MoveL Offs(p0,121.96290000000002,30.827499999999997, 0), v100, z5, tool0;
MoveL Offs(p0,122.3,29.7, 0), v100, z5, tool0;
MoveL Offs(p0,121.74480000000001,29.45120000000001, 0), v100, z5, tool0;
MoveL Offs(p0,121.0427,29.323799999999995, 0), v100, z5, tool0;
MoveL Offs(p0,120.0904,29.197600000000005, 0), v100, z5, tool0;
MoveL Offs(p0,118.9125,29.075, 0), v100, z5, tool0;
MoveL Offs(p0,117.5336,28.9584, 0), v100, z5, tool0;
MoveL Offs(p0,115.97829999999999,28.8502, 0), v100, z5, tool0;
MoveL Offs(p0,114.2712,28.7528, 0), v100, z5, tool0;
MoveL Offs(p0,112.4369,28.668600000000005, 0), v100, z5, tool0;
MoveL Offs(p0,110.5,28.6, 0), v100, z5, tool0;
MoveL Offs(p0,103.26039999999998,28.309299999999997, 0), v100, z5, tool0;
MoveL Offs(p0,101.38480000000001,28.1456, 0), v100, z5, tool0;
MoveL Offs(p0,99.7,27.9375, 0), v100, z5, tool0;
MoveL Offs(p0,98.1592,27.6784, 0), v100, z5, tool0;
MoveL Offs(p0,96.7156,27.361699999999995, 0), v100, z5, tool0;
MoveL Offs(p0,95.32240000000002,26.9808, 0), v100, z5, tool0;
MoveL Offs(p0,93.9328,26.5291, 0), v100, z5, tool0;
MoveL Offs(p0,92.5,26.0, 0), v100, z5, tool0;
MoveL Offs(p0,91.52130000000001,25.629400000000004, 0), v100, z5, tool0;
MoveL Offs(p0,90.57440000000004,25.24320000000001, 0), v100, z5, tool0;
MoveL Offs(p0,89.6731,24.8498, 0), v100, z5, tool0;
MoveL Offs(p0,88.83120000000001,24.4576, 0), v100, z5, tool0;
MoveL Offs(p0,88.0625,24.075, 0), v100, z5, tool0;
MoveL Offs(p0,87.3808,23.7104, 0), v100, z5, tool0;
MoveL Offs(p0,86.79990000000001,23.3722, 0), v100, z5, tool0;
MoveL Offs(p0,86.3336,23.068800000000003, 0), v100, z5, tool0;
MoveL Offs(p0,85.99570000000001,22.808600000000002, 0), v100, z5, tool0;
MoveL Offs(p0,85.8,22.6, 0), v100, z5, tool0;
MoveL Offs(p0,85.14040000000001,22.216700000000003, 0), v100, z5, tool0;
MoveL Offs(p0,83.57879999999997,23.8249, 0), v100, z5, tool0;
MoveL Offs(p0,82.7536,25.5728, 0), v100, z5, tool0;
MoveL Offs(p0,81.95,27.7875, 0), v100, z5, tool0;
MoveL Offs(p0,81.2064,30.347199999999997, 0), v100, z5, tool0;
MoveL Offs(p0,80.56120000000001,33.130100000000006, 0), v100, z5, tool0;
MoveL Offs(p0,80.0528,36.0144, 0), v100, z5, tool0;
MoveL Offs(p0,79.7196,38.8783, 0), v100, z5, tool0;
MoveL Offs(p0,79.6,41.6, 0), v100, z5, tool0;
MoveL Offs(p0,80.06560000000002,47.246400000000015, 0), v100, z5, tool0;
MoveL Offs(p0,80.61339999999998,49.9151, 0), v100, z5, tool0;
MoveL Offs(p0,81.3808,52.49920000000001, 0), v100, z5, tool0;
MoveL Offs(p0,82.375,55.0125, 0), v100, z5, tool0;
MoveL Offs(p0,83.6032,57.46880000000001, 0), v100, z5, tool0;
MoveL Offs(p0,85.0726,59.88190000000001, 0), v100, z5, tool0;
MoveL Offs(p0,86.7904,62.265600000000006, 0), v100, z5, tool0;
MoveL Offs(p0,88.7638,64.6337, 0), v100, z5, tool0;
MoveL Offs(p0,91.0,67.0, 0), v100, z5, tool0;
MoveL Offs(p0,93.10790000000001,69.02610000000001, 0), v100, z5, tool0;
MoveL Offs(p0,95.17920000000002,70.84880000000001, 0), v100, z5, tool0;
MoveL Offs(p0,97.2253,72.4747, 0), v100, z5, tool0;
MoveL Offs(p0,99.2576,73.91040000000001, 0), v100, z5, tool0;
MoveL Offs(p0,101.2875,75.1625, 0), v100, z5, tool0;
MoveL Offs(p0,103.32639999999999,76.2376, 0), v100, z5, tool0;
MoveL Offs(p0,105.3857,77.1423, 0), v100, z5, tool0;
MoveL Offs(p0,107.4768,77.88320000000002, 0), v100, z5, tool0;
MoveL Offs(p0,109.6111,78.4669, 0), v100, z5, tool0;
MoveL Offs(p0,111.8,78.9, 0), v100, z5, tool0;
MoveL Offs(p0,114.63920000000005,79.21440000000003, 0), v100, z5, tool0;
MoveL Offs(p0,116.24330000000002,79.2951, 0), v100, z5, tool0;
MoveL Offs(p0,117.8816,79.3272, 0), v100, z5, tool0;
MoveL Offs(p0,119.4875,79.3125, 0), v100, z5, tool0;
MoveL Offs(p0,120.9944,79.25280000000001, 0), v100, z5, tool0;
MoveL Offs(p0,122.3357,79.1499, 0), v100, z5, tool0;
MoveL Offs(p0,124.7,78.6, 0), v100, z5, tool0;
MoveL Offs(p0,124.7,78.6, 0), v100, z5, tool0;
MoveJ Offs(p0,158.3,63.6, 10), v100, z1, tool0;
MoveL Offs(p0,158.5876,62.95320000000002, 0), v100, z5, tool0;
MoveL Offs(p0,158.84880000000007,62.33760000000001, 0), v100, z5, tool0;
MoveL Offs(p0,159.0812,61.76039999999999, 0), v100, z5, tool0;
MoveL Offs(p0,159.2824,61.2288, 0), v100, z5, tool0;
MoveL Offs(p0,159.45,60.75, 0), v100, z5, tool0;
MoveL Offs(p0,159.5816,60.3312, 0), v100, z5, tool0;
MoveL Offs(p0,159.6748,59.979600000000005, 0), v100, z5, tool0;
MoveL Offs(p0,159.7272,59.70240000000001, 0), v100, z5, tool0;
MoveL Offs(p0,159.7364,59.5068, 0), v100, z5, tool0;
MoveL Offs(p0,159.7,59.4, 0), v100, z5, tool0;
MoveL Offs(p0,158.64339999999999,59.0742, 0), v100, z5, tool0;
MoveL Offs(p0,157.9128,58.9104, 0), v100, z5, tool0;
MoveL Offs(p0,157.025,58.725, 0), v100, z5, tool0;
MoveL Offs(p0,155.9992,58.5216, 0), v100, z5, tool0;
MoveL Offs(p0,154.85459999999998,58.3038, 0), v100, z5, tool0;
MoveL Offs(p0,153.6104,58.07520000000001, 0), v100, z5, tool0;
MoveL Offs(p0,152.28580000000002,57.8394, 0), v100, z5, tool0;
MoveL Offs(p0,150.9,57.6, 0), v100, z5, tool0;
MoveL Offs(p0,147.34920000000002,57.077, 0), v100, z5, tool0;
MoveL Offs(p0,143.98560000000003,56.764000000000024, 0), v100, z5, tool0;
MoveL Offs(p0,140.8524,56.654999999999994, 0), v100, z5, tool0;
MoveL Offs(p0,137.99280000000002,56.74400000000001, 0), v100, z5, tool0;
MoveL Offs(p0,135.45,57.025, 0), v100, z5, tool0;
MoveL Offs(p0,131.4876,58.138999999999996, 0), v100, z5, tool0;
MoveL Offs(p0,130.1544,58.96, 0), v100, z5, tool0;
MoveL Offs(p0,129.3108,59.949, 0), v100, z5, tool0;
MoveL Offs(p0,129.0,61.1, 0), v100, z5, tool0;
MoveL Offs(p0,129.3213,61.807399999999994, 0), v100, z5, tool0;
MoveL Offs(p0,129.55360000000002,62.20880000000001, 0), v100, z5, tool0;
MoveL Offs(p0,129.8375,62.675, 0), v100, z5, tool0;
MoveL Offs(p0,130.1664,63.1952, 0), v100, z5, tool0;
MoveL Offs(p0,130.5337,63.7586, 0), v100, z5, tool0;
MoveL Offs(p0,130.9328,64.35440000000001, 0), v100, z5, tool0;
MoveL Offs(p0,131.3571,64.9718, 0), v100, z5, tool0;
MoveL Offs(p0,131.8,65.6, 0), v100, z5, tool0;
MoveL Offs(p0,132.95589999999999,67.0506, 0), v100, z5, tool0;
MoveL Offs(p0,134.25520000000006,68.45680000000002, 0), v100, z5, tool0;
MoveL Offs(p0,135.68529999999998,69.81020000000001, 0), v100, z5, tool0;
MoveL Offs(p0,137.23360000000002,71.10240000000002, 0), v100, z5, tool0;
MoveL Offs(p0,138.8875,72.325, 0), v100, z5, tool0;
MoveL Offs(p0,140.6344,73.4696, 0), v100, z5, tool0;
MoveL Offs(p0,142.4617,74.5278, 0), v100, z5, tool0;
MoveL Offs(p0,144.35680000000002,75.4912, 0), v100, z5, tool0;
MoveL Offs(p0,146.30710000000002,76.35140000000001, 0), v100, z5, tool0;
MoveL Offs(p0,148.3,77.1, 0), v100, z5, tool0;
MoveL Offs(p0,153.5,78.9, 0), v100, z5, tool0;
MoveL Offs(p0,155.1,73.2, 0), v100, z5, tool0;
MoveL Offs(p0,155.35970000000003,72.2346, 0), v100, z5, tool0;
MoveL Offs(p0,155.65360000000004,71.21280000000002, 0), v100, z5, tool0;
MoveL Offs(p0,155.9739,70.1562, 0), v100, z5, tool0;
MoveL Offs(p0,156.3128,69.0864, 0), v100, z5, tool0;
MoveL Offs(p0,156.6625,68.025, 0), v100, z5, tool0;
MoveL Offs(p0,157.0152,66.9936, 0), v100, z5, tool0;
MoveL Offs(p0,157.36309999999997,66.0138, 0), v100, z5, tool0;
MoveL Offs(p0,157.69840000000002,65.1072, 0), v100, z5, tool0;
MoveL Offs(p0,158.01330000000002,64.2954, 0), v100, z5, tool0;
MoveL Offs(p0,158.3,63.6, 0), v100, z5, tool0;
MoveL Offs(p0,158.3,63.6, 0), v100, z5, tool0;
MoveJ Offs(p0,118.3,63.5, 10), v100, z1, tool0;
MoveL Offs(p0,118.0768,57.86959999999999, 0), v100, z5, tool0;
MoveL Offs(p0,118.04589999999999,56.6078, 0), v100, z5, tool0;
MoveL Offs(p0,118.0216,55.31120000000001, 0), v100, z5, tool0;
MoveL Offs(p0,118.0057,54.001400000000004, 0), v100, z5, tool0;
MoveL Offs(p0,118.0,52.7, 0), v100, z5, tool0;
MoveL Offs(p0,117.9,44.9, 0), v100, z5, tool0;
MoveL Offs(p0,115.2,45.4, 0), v100, z5, tool0;
MoveL Offs(p0,113.98960000000004,45.60160000000002, 0), v100, z5, tool0;
MoveL Offs(p0,113.1804,45.7159, 0), v100, z5, tool0;
MoveL Offs(p0,112.26080000000002,45.83680000000001, 0), v100, z5, tool0;
MoveL Offs(p0,111.25,45.9625, 0), v100, z5, tool0;
MoveL Offs(p0,110.16720000000001,46.0912, 0), v100, z5, tool0;
MoveL Offs(p0,109.0316,46.2211, 0), v100, z5, tool0;
MoveL Offs(p0,107.86240000000001,46.3504, 0), v100, z5, tool0;
MoveL Offs(p0,106.6788,46.4773, 0), v100, z5, tool0;
MoveL Offs(p0,105.5,46.6, 0), v100, z5, tool0;
MoveL Offs(p0,100.6179,47.25800000000001, 0), v100, z5, tool0;
MoveL Offs(p0,96.65920000000001,48.192000000000014, 0), v100, z5, tool0;
MoveL Offs(p0,93.6353,49.372, 0), v100, z5, tool0;
MoveL Offs(p0,91.55760000000001,50.768, 0), v100, z5, tool0;
MoveL Offs(p0,90.4375,52.35, 0), v100, z5, tool0;
MoveL Offs(p0,90.28639999999999,54.088, 0), v100, z5, tool0;
MoveL Offs(p0,91.11569999999999,55.952, 0), v100, z5, tool0;
MoveL Offs(p0,92.9368,57.912, 0), v100, z5, tool0;
MoveL Offs(p0,95.7611,59.93800000000001, 0), v100, z5, tool0;
MoveL Offs(p0,99.6,62.0, 0), v100, z5, tool0;
MoveL Offs(p0,101.475,62.868600000000015, 0), v100, z5, tool0;
MoveL Offs(p0,103.41600000000001,63.66880000000002, 0), v100, z5, tool0;
MoveL Offs(p0,105.38699999999999,64.39219999999999, 0), v100, z5, tool0;
MoveL Offs(p0,107.35200000000002,65.03040000000001, 0), v100, z5, tool0;
MoveL Offs(p0,109.275,65.575, 0), v100, z5, tool0;
MoveL Offs(p0,111.12,66.0176, 0), v100, z5, tool0;
MoveL Offs(p0,112.851,66.3498, 0), v100, z5, tool0;
MoveL Offs(p0,114.43200000000002,66.56320000000001, 0), v100, z5, tool0;
MoveL Offs(p0,115.827,66.6494, 0), v100, z5, tool0;
MoveL Offs(p0,117.0,66.6, 0), v100, z5, tool0;
MoveL Offs(p0,117.74069999999999,66.2643, 0), v100, z5, tool0;
MoveL Offs(p0,117.91839999999999,66.04159999999999, 0), v100, z5, tool0;
MoveL Offs(p0,118.0625,65.7625, 0), v100, z5, tool0;
MoveL Offs(p0,118.1736,65.4264, 0), v100, z5, tool0;
MoveL Offs(p0,118.25230000000002,65.0327, 0), v100, z5, tool0;
MoveL Offs(p0,118.29920000000001,64.5808, 0), v100, z5, tool0;
MoveL Offs(p0,118.31490000000001,64.0701, 0), v100, z5, tool0;
MoveL Offs(p0,118.3,63.5, 0), v100, z5, tool0;
MoveL Offs(p0,118.3,63.5, 0), v100, z5, tool0;
MoveJ Offs(p0,77.2,61.7, 10), v100, z1, tool0;
MoveL Offs(p0,80.9,60.2, 0), v100, z5, tool0;
MoveL Offs(p0,78.9,55.1, 0), v100, z5, tool0;
MoveL Offs(p0,78.6038,54.2505, 0), v100, z5, tool0;
MoveL Offs(p0,78.31840000000001,53.39200000000002, 0), v100, z5, tool0;
MoveL Offs(p0,78.0486,52.5395, 0), v100, z5, tool0;
MoveL Offs(p0,77.7992,51.708000000000006, 0), v100, z5, tool0;
MoveL Offs(p0,77.575,50.9125, 0), v100, z5, tool0;
MoveL Offs(p0,77.3808,50.168, 0), v100, z5, tool0;
MoveL Offs(p0,77.22139999999999,49.4895, 0), v100, z5, tool0;
MoveL Offs(p0,77.1016,48.892, 0), v100, z5, tool0;
MoveL Offs(p0,77.02619999999999,48.39050000000001, 0), v100, z5, tool0;
MoveL Offs(p0,77.0,48.0, 0), v100, z5, tool0;
MoveL Offs(p0,76.732,46.63440000000001, 0), v100, z5, tool0;
MoveL Offs(p0,76.37899999999999,46.28009999999999, 0), v100, z5, tool0;
MoveL Offs(p0,75.864,46.147200000000005, 0), v100, z5, tool0;
MoveL Offs(p0,75.175,46.2375, 0), v100, z5, tool0;
MoveL Offs(p0,74.3,46.5528, 0), v100, z5, tool0;
MoveL Offs(p0,73.227,47.09490000000001, 0), v100, z5, tool0;
MoveL Offs(p0,70.439,48.8667, 0), v100, z5, tool0;
MoveL Offs(p0,68.7,50.1, 0), v100, z5, tool0;
MoveL Offs(p0,67.0042,51.4408, 0), v100, z5, tool0;
MoveL Offs(p0,65.46560000000002,52.810400000000016, 0), v100, z5, tool0;
MoveL Offs(p0,64.0974,54.1896, 0), v100, z5, tool0;
MoveL Offs(p0,62.91279999999999,55.5592, 0), v100, z5, tool0;
MoveL Offs(p0,61.925,56.9, 0), v100, z5, tool0;
MoveL Offs(p0,61.1472,58.1928, 0), v100, z5, tool0;
MoveL Offs(p0,60.59259999999999,59.4184, 0), v100, z5, tool0;
MoveL Offs(p0,60.2744,60.5576, 0), v100, z5, tool0;
MoveL Offs(p0,60.205799999999996,61.5912, 0), v100, z5, tool0;
MoveL Offs(p0,60.4,62.5, 0), v100, z5, tool0;
MoveL Offs(p0,60.80080000000002,63.24960000000002, 0), v100, z5, tool0;
MoveL Offs(p0,61.10920000000001,63.5179, 0), v100, z5, tool0;
MoveL Offs(p0,61.51840000000001,63.7208, 0), v100, z5, tool0;
MoveL Offs(p0,62.05,63.8625, 0), v100, z5, tool0;
MoveL Offs(p0,62.7256,63.947199999999995, 0), v100, z5, tool0;
MoveL Offs(p0,63.5668,63.9791, 0), v100, z5, tool0;
MoveL Offs(p0,64.5952,63.9624, 0), v100, z5, tool0;
MoveL Offs(p0,65.8324,63.901300000000006, 0), v100, z5, tool0;
MoveL Offs(p0,67.3,63.8, 0), v100, z5, tool0;
MoveL Offs(p0,69.44320000000002,63.55280000000001, 0), v100, z5, tool0;
MoveL Offs(p0,70.55980000000001,63.3842, 0), v100, z5, tool0;
MoveL Offs(p0,71.67760000000001,63.19040000000001, 0), v100, z5, tool0;
MoveL Offs(p0,72.775,62.975, 0), v100, z5, tool0;
MoveL Offs(p0,73.8304,62.74159999999999, 0), v100, z5, tool0;
MoveL Offs(p0,74.8222,62.4938, 0), v100, z5, tool0;
MoveL Offs(p0,75.7288,62.235200000000006, 0), v100, z5, tool0;
MoveL Offs(p0,76.52860000000001,61.96939999999999, 0), v100, z5, tool0;
MoveL Offs(p0,77.2,61.7, 0), v100, z5, tool0;
MoveL Offs(p0,77.2,61.7, 0), v100, z5, tool0;
MoveJ Offs(p0,252.7,48.8, 10), v100, z1, tool0;
MoveL Offs(p0,252.4381,48.368900000000004, 0), v100, z5, tool0;
MoveL Offs(p0,252.35920000000002,48.348800000000004, 0), v100, z5, tool0;
MoveL Offs(p0,252.2875,48.3875, 0), v100, z5, tool0;
MoveL Offs(p0,252.22479999999996,48.4832, 0), v100, z5, tool0;
MoveL Offs(p0,252.1087,49.0943, 0), v100, z5, tool0;
MoveL Offs(p0,252.1,49.4, 0), v100, z5, tool0;
MoveL Offs(p0,252.3408,50.8035, 0), v100, z5, tool0;
MoveL Offs(p0,252.4232,50.824000000000005, 0), v100, z5, tool0;
MoveL Offs(p0,252.51040000000003,50.79050000000001, 0), v100, z5, tool0;
MoveL Offs(p0,252.6,50.7, 0), v100, z5, tool0;
MoveL Offs(p0,252.81059999999997,50.28959999999999, 0), v100, z5, tool0;
MoveL Offs(p0,252.85119999999998,50.10320000000001, 0), v100, z5, tool0;
MoveL Offs(p0,252.875,49.9, 0), v100, z5, tool0;
MoveL Offs(p0,252.8808,49.6848, 0), v100, z5, tool0;
MoveL Offs(p0,252.8674,49.4624, 0), v100, z5, tool0;
MoveL Offs(p0,252.83360000000002,49.2376, 0), v100, z5, tool0;
MoveL Offs(p0,252.7,48.8, 0), v100, z5, tool0;
MoveJ Offs(p0,184.5,39.8, 10), v100, z1, tool0;
MoveL Offs(p0,186.67090000000002,39.054300000000005, 0), v100, z5, tool0;
MoveL Offs(p0,188.60720000000006,38.43040000000001, 0), v100, z5, tool0;
MoveL Offs(p0,190.3743,37.918099999999995, 0), v100, z5, tool0;
MoveL Offs(p0,192.0376,37.5072, 0), v100, z5, tool0;
MoveL Offs(p0,193.6625,37.1875, 0), v100, z5, tool0;
MoveL Offs(p0,195.3144,36.9488, 0), v100, z5, tool0;
MoveL Offs(p0,197.0587,36.780899999999995, 0), v100, z5, tool0;
MoveL Offs(p0,198.9608,36.67360000000001, 0), v100, z5, tool0;
MoveL Offs(p0,201.0861,36.6167, 0), v100, z5, tool0;
MoveL Offs(p0,203.5,36.6, 0), v100, z5, tool0;
MoveL Offs(p0,213.5728,36.852, 0), v100, z5, tool0;
MoveL Offs(p0,215.03040000000001,36.953500000000005, 0), v100, z5, tool0;
MoveL Offs(p0,216.34160000000003,37.06400000000001, 0), v100, z5, tool0;
MoveL Offs(p0,217.4752,37.1805, 0), v100, z5, tool0;
MoveL Offs(p0,218.4,37.3, 0), v100, z5, tool0;
MoveL Offs(p0,223.2,38.2, 0), v100, z5, tool0;
MoveL Offs(p0,220.2,33.8, 0), v100, z5, tool0;
MoveL Offs(p0,218.2322,31.121900000000004, 0), v100, z5, tool0;
MoveL Offs(p0,216.1576000000001,28.599200000000007, 0), v100, z5, tool0;
MoveL Offs(p0,213.95940000000002,26.219299999999997, 0), v100, z5, tool0;
MoveL Offs(p0,211.6208,23.9696, 0), v100, z5, tool0;
MoveL Offs(p0,209.125,21.8375, 0), v100, z5, tool0;
MoveL Offs(p0,206.45519999999996,19.810399999999998, 0), v100, z5, tool0;
MoveL Offs(p0,203.59459999999999,17.8757, 0), v100, z5, tool0;
MoveL Offs(p0,200.52640000000002,16.0208, 0), v100, z5, tool0;
MoveL Offs(p0,197.2338,14.233100000000002, 0), v100, z5, tool0;
MoveL Offs(p0,193.7,12.5, 0), v100, z5, tool0;
MoveL Offs(p0,189.09650000000005,10.568900000000001, 0), v100, z5, tool0;
MoveL Offs(p0,184.28000000000006,8.979200000000002, 0), v100, z5, tool0;
MoveL Offs(p0,179.33149999999998,7.736299999999998, 0), v100, z5, tool0;
MoveL Offs(p0,174.33200000000002,6.8456, 0), v100, z5, tool0;
MoveL Offs(p0,169.3625,6.3125, 0), v100, z5, tool0;
MoveL Offs(p0,164.504,6.1424, 0), v100, z5, tool0;
MoveL Offs(p0,159.8375,6.3407, 0), v100, z5, tool0;
MoveL Offs(p0,155.44400000000002,6.912800000000002, 0), v100, z5, tool0;
MoveL Offs(p0,151.4045,7.8641000000000005, 0), v100, z5, tool0;
MoveL Offs(p0,147.8,9.2, 0), v100, z5, tool0;
MoveL Offs(p0,145.62860000000003,10.322400000000002, 0), v100, z5, tool0;
MoveL Offs(p0,143.36480000000003,11.723200000000004, 0), v100, z5, tool0;
MoveL Offs(p0,141.08419999999998,13.3328, 0), v100, z5, tool0;
MoveL Offs(p0,138.8624,15.0816, 0), v100, z5, tool0;
MoveL Offs(p0,136.775,16.9, 0), v100, z5, tool0;
MoveL Offs(p0,134.8976,18.7184, 0), v100, z5, tool0;
MoveL Offs(p0,133.3058,20.4672, 0), v100, z5, tool0;
MoveL Offs(p0,132.0752,22.076800000000002, 0), v100, z5, tool0;
MoveL Offs(p0,131.28140000000002,23.477600000000002, 0), v100, z5, tool0;
MoveL Offs(p0,131.0,24.6, 0), v100, z5, tool0;
MoveL Offs(p0,131.37480000000002,26.3772, 0), v100, z5, tool0;
MoveL Offs(p0,132.4504,28.257600000000007, 0), v100, z5, tool0;
MoveL Offs(p0,134.1536,30.194399999999995, 0), v100, z5, tool0;
MoveL Offs(p0,136.4112,32.1408, 0), v100, z5, tool0;
MoveL Offs(p0,139.15,34.05, 0), v100, z5, tool0;
MoveL Offs(p0,142.29680000000002,35.8752, 0), v100, z5, tool0;
MoveL Offs(p0,145.7784,37.5696, 0), v100, z5, tool0;
MoveL Offs(p0,149.52160000000003,39.086400000000005, 0), v100, z5, tool0;
MoveL Offs(p0,153.4532,40.3788, 0), v100, z5, tool0;
MoveL Offs(p0,157.5,41.4, 0), v100, z5, tool0;
MoveL Offs(p0,160.7049,42.01130000000001, 0), v100, z5, tool0;
MoveL Offs(p0,163.63920000000005,42.46240000000001, 0), v100, z5, tool0;
MoveL Offs(p0,166.3623,42.74909999999999, 0), v100, z5, tool0;
MoveL Offs(p0,168.93359999999998,42.867200000000004, 0), v100, z5, tool0;
MoveL Offs(p0,171.4125,42.8125, 0), v100, z5, tool0;
MoveL Offs(p0,173.85840000000002,42.580799999999996, 0), v100, z5, tool0;
MoveL Offs(p0,176.33069999999998,42.167899999999996, 0), v100, z5, tool0;
MoveL Offs(p0,181.59210000000002,40.7817, 0), v100, z5, tool0;
MoveL Offs(p0,184.5,39.8, 0), v100, z5, tool0;
MoveL Offs(p0,184.5,39.8, 0), v100, z5, tool0;
MoveJ Offs(p0,67.2,31.3, 10), v100, z1, tool0;
MoveL Offs(p0,69.19580000000002,30.4745, 0), v100, z5, tool0;
MoveL Offs(p0,71.10640000000002,29.556000000000004, 0), v100, z5, tool0;
MoveL Offs(p0,72.9366,28.541500000000003, 0), v100, z5, tool0;
MoveL Offs(p0,74.69120000000001,27.427999999999997, 0), v100, z5, tool0;
MoveL Offs(p0,76.375,26.2125, 0), v100, z5, tool0;
MoveL Offs(p0,77.99280000000002,24.892000000000003, 0), v100, z5, tool0;
MoveL Offs(p0,79.54939999999999,23.4635, 0), v100, z5, tool0;
MoveL Offs(p0,81.04960000000001,21.924, 0), v100, z5, tool0;
MoveL Offs(p0,82.49820000000001,20.2705, 0), v100, z5, tool0;
MoveL Offs(p0,83.9,18.5, 0), v100, z5, tool0;
MoveL Offs(p0,88.2,12.8, 0), v100, z5, tool0;
MoveL Offs(p0,84.9,13.5, 0), v100, z5, tool0;
MoveL Offs(p0,82.76840000000001,14.0779, 0), v100, z5, tool0;
MoveL Offs(p0,80.23120000000003,14.991200000000003, 0), v100, z5, tool0;
MoveL Offs(p0,77.4048,16.1793, 0), v100, z5, tool0;
MoveL Offs(p0,74.4056,17.5816, 0), v100, z5, tool0;
MoveL Offs(p0,71.35,19.1375, 0), v100, z5, tool0;
MoveL Offs(p0,68.3544,20.7864, 0), v100, z5, tool0;
MoveL Offs(p0,65.5352,22.4677, 0), v100, z5, tool0;
MoveL Offs(p0,63.00880000000001,24.120800000000003, 0), v100, z5, tool0;
MoveL Offs(p0,60.891600000000004,25.6851, 0), v100, z5, tool0;
MoveL Offs(p0,59.3,27.1, 0), v100, z5, tool0;
MoveL Offs(p0,58.605100000000014,27.788100000000007, 0), v100, z5, tool0;
MoveL Offs(p0,57.96480000000001,28.464800000000007, 0), v100, z5, tool0;
MoveL Offs(p0,57.38570000000001,29.1187, 0), v100, z5, tool0;
MoveL Offs(p0,56.874400000000016,29.738400000000002, 0), v100, z5, tool0;
MoveL Offs(p0,56.4375,30.3125, 0), v100, z5, tool0;
MoveL Offs(p0,56.0816,30.829600000000006, 0), v100, z5, tool0;
MoveL Offs(p0,55.813300000000005,31.278299999999994, 0), v100, z5, tool0;
MoveL Offs(p0,55.6392,31.647200000000005, 0), v100, z5, tool0;
MoveL Offs(p0,55.56590000000001,31.9249, 0), v100, z5, tool0;
MoveL Offs(p0,55.6,32.1, 0), v100, z5, tool0;
MoveL Offs(p0,56.01930000000002,32.46640000000001, 0), v100, z5, tool0;
MoveL Offs(p0,56.710400000000014,32.72720000000001, 0), v100, z5, tool0;
MoveL Offs(p0,57.63309999999999,32.8848, 0), v100, z5, tool0;
MoveL Offs(p0,58.74720000000001,32.9416, 0), v100, z5, tool0;
MoveL Offs(p0,60.0125,32.9, 0), v100, z5, tool0;
MoveL Offs(p0,61.3888,32.7624, 0), v100, z5, tool0;
MoveL Offs(p0,62.8359,32.5312, 0), v100, z5, tool0;
MoveL Offs(p0,65.7817,31.7976, 0), v100, z5, tool0;
MoveL Offs(p0,67.2,31.3, 0), v100, z5, tool0;
MoveL Offs(p0,67.2,31.3, 0), v100, z5, tool0;
MoveJ Offs(p0,122.7,24.5, 10), v100, z1, tool0;
MoveL Offs(p0,123.38410000000002,24.163500000000006, 0), v100, z5, tool0;
MoveL Offs(p0,124.16480000000006,23.704000000000004, 0), v100, z5, tool0;
MoveL Offs(p0,125.02470000000001,23.1365, 0), v100, z5, tool0;
MoveL Offs(p0,125.94640000000001,22.476000000000003, 0), v100, z5, tool0;
MoveL Offs(p0,126.9125,21.7375, 0), v100, z5, tool0;
MoveL Offs(p0,127.9056,20.935999999999996, 0), v100, z5, tool0;
MoveL Offs(p0,128.9083,20.086499999999997, 0), v100, z5, tool0;
MoveL Offs(p0,129.90320000000003,19.204, 0), v100, z5, tool0;
MoveL Offs(p0,130.87290000000002,18.303500000000003, 0), v100, z5, tool0;
MoveL Offs(p0,131.8,17.4, 0), v100, z5, tool0;
MoveL Offs(p0,132.74150000000003,16.479000000000003, 0), v100, z5, tool0;
MoveL Offs(p0,133.75200000000004,15.528000000000006, 0), v100, z5, tool0;
MoveL Offs(p0,134.8105,14.564999999999998, 0), v100, z5, tool0;
MoveL Offs(p0,135.89600000000002,13.607999999999999, 0), v100, z5, tool0;
MoveL Offs(p0,136.9875,12.675, 0), v100, z5, tool0;
MoveL Offs(p0,138.06400000000002,11.783999999999999, 0), v100, z5, tool0;
MoveL Offs(p0,139.1045,10.953, 0), v100, z5, tool0;
MoveL Offs(p0,140.08800000000002,10.2, 0), v100, z5, tool0;
MoveL Offs(p0,140.9935,9.543000000000001, 0), v100, z5, tool0;
MoveL Offs(p0,141.8,9.0, 0), v100, z5, tool0;
MoveL Offs(p0,142.66990000000004,8.4539, 0), v100, z5, tool0;
MoveL Offs(p0,143.41920000000002,7.955200000000002, 0), v100, z5, tool0;
MoveL Offs(p0,144.0473,7.5033, 0), v100, z5, tool0;
MoveL Offs(p0,144.55360000000002,7.0976, 0), v100, z5, tool0;
MoveL Offs(p0,144.9375,6.7375, 0), v100, z5, tool0;
MoveL Offs(p0,145.1984,6.422399999999999, 0), v100, z5, tool0;
MoveL Offs(p0,145.3357,6.1517, 0), v100, z5, tool0;
MoveL Offs(p0,145.34880000000004,5.9248, 0), v100, z5, tool0;
MoveL Offs(p0,145.2371,5.7411, 0), v100, z5, tool0;
MoveL Offs(p0,145.0,5.6, 0), v100, z5, tool0;
MoveL Offs(p0,141.8641,4.6761, 0), v100, z5, tool0;
MoveL Offs(p0,138.48880000000003,3.9448000000000016, 0), v100, z5, tool0;
MoveL Offs(p0,134.9227,3.4067, 0), v100, z5, tool0;
MoveL Offs(p0,131.2144,3.0624000000000002, 0), v100, z5, tool0;
MoveL Offs(p0,127.4125,2.9125, 0), v100, z5, tool0;
MoveL Offs(p0,123.56559999999999,2.9576000000000002, 0), v100, z5, tool0;
MoveL Offs(p0,119.72229999999999,3.1983000000000006, 0), v100, z5, tool0;
MoveL Offs(p0,115.93119999999999,3.6352, 0), v100, z5, tool0;
MoveL Offs(p0,112.24090000000001,4.2689, 0), v100, z5, tool0;
MoveL Offs(p0,108.7,5.1, 0), v100, z5, tool0;
MoveL Offs(p0,106.14359999999999,5.89, 0), v100, z5, tool0;
MoveL Offs(p0,103.54880000000003,6.860000000000002, 0), v100, z5, tool0;
MoveL Offs(p0,100.96719999999999,7.980000000000001, 0), v100, z5, tool0;
MoveL Offs(p0,98.4504,9.22, 0), v100, z5, tool0;
MoveL Offs(p0,96.05,10.55, 0), v100, z5, tool0;
MoveL Offs(p0,93.8176,11.940000000000001, 0), v100, z5, tool0;
MoveL Offs(p0,91.8048,13.36, 0), v100, z5, tool0;
MoveL Offs(p0,90.06320000000001,14.780000000000001, 0), v100, z5, tool0;
MoveL Offs(p0,88.64439999999999,16.17, 0), v100, z5, tool0;
MoveL Offs(p0,87.6,17.5, 0), v100, z5, tool0;
MoveL Offs(p0,87.196,18.130600000000005, 0), v100, z5, tool0;
MoveL Offs(p0,86.88800000000002,18.656800000000008, 0), v100, z5, tool0;
MoveL Offs(p0,86.68199999999999,19.1002, 0), v100, z5, tool0;
MoveL Offs(p0,86.584,19.482400000000005, 0), v100, z5, tool0;
MoveL Offs(p0,86.6,19.825, 0), v100, z5, tool0;
MoveL Offs(p0,86.736,20.1496, 0), v100, z5, tool0;
MoveL Offs(p0,86.998,20.4778, 0), v100, z5, tool0;
MoveL Offs(p0,87.39200000000001,20.831200000000003, 0), v100, z5, tool0;
MoveL Offs(p0,87.924,21.2314, 0), v100, z5, tool0;
MoveL Offs(p0,88.6,21.7, 0), v100, z5, tool0;
MoveL Offs(p0,89.9469,22.4737, 0), v100, z5, tool0;
MoveL Offs(p0,91.46720000000002,23.173600000000008, 0), v100, z5, tool0;
MoveL Offs(p0,93.1603,23.7979, 0), v100, z5, tool0;
MoveL Offs(p0,95.02560000000003,24.3448, 0), v100, z5, tool0;
MoveL Offs(p0,97.0625,24.8125, 0), v100, z5, tool0;
MoveL Offs(p0,99.2704,25.1992, 0), v100, z5, tool0;
MoveL Offs(p0,101.6487,25.503099999999996, 0), v100, z5, tool0;
MoveL Offs(p0,104.19680000000001,25.722400000000004, 0), v100, z5, tool0;
MoveL Offs(p0,106.9141,25.8553, 0), v100, z5, tool0;
MoveL Offs(p0,109.8,25.9, 0), v100, z5, tool0;
MoveL Offs(p0,117.675,25.6125, 0), v100, z5, tool0;
MoveL Offs(p0,118.90799999999999,25.4536, 0), v100, z5, tool0;
MoveL Offs(p0,120.027,25.2623, 0), v100, z5, tool0;
MoveL Offs(p0,121.03200000000001,25.0392, 0), v100, z5, tool0;
MoveL Offs(p0,121.923,24.7849, 0), v100, z5, tool0;
MoveL Offs(p0,122.7,24.5, 0), v100, z5, tool0;
MoveL Offs(p0,122.7,24.5, 0), v100, z5, tool0;
MoveJ Offs(p0,368.6,345.8, 10), v100, z1, tool0;
MoveL Offs(p0,368.82320000000016,345.5480000000001, 0), v100, z5, tool0;
MoveL Offs(p0,368.9618,345.4579999999999, 0), v100, z5, tool0;
MoveL Offs(p0,369.1136,345.392, 0), v100, z5, tool0;
MoveL Offs(p0,369.275,345.35, 0), v100, z5, tool0;
MoveL Offs(p0,369.4424,345.332, 0), v100, z5, tool0;
MoveL Offs(p0,369.6122,345.338, 0), v100, z5, tool0;
MoveL Offs(p0,369.78080000000006,345.36800000000005, 0), v100, z5, tool0;
MoveL Offs(p0,369.94460000000004,345.422, 0), v100, z5, tool0;
MoveL Offs(p0,370.1,345.5, 0), v100, z5, tool0;
MoveL Offs(p0,370.44500000000005,345.7523, 0), v100, z5, tool0;
MoveL Offs(p0,370.70000000000005,345.97040000000004, 0), v100, z5, tool0;
MoveL Offs(p0,370.865,346.1560999999999, 0), v100, z5, tool0;
MoveL Offs(p0,370.94,346.3112, 0), v100, z5, tool0;
MoveL Offs(p0,370.925,346.4375, 0), v100, z5, tool0;
MoveL Offs(p0,370.82,346.53679999999997, 0), v100, z5, tool0;
MoveL Offs(p0,370.625,346.6109, 0), v100, z5, tool0;
MoveL Offs(p0,370.34000000000003,346.6616, 0), v100, z5, tool0;
MoveL Offs(p0,369.5,346.7, 0), v100, z5, tool0;
MoveL Offs(p0,368.6375,346.4375, 0), v100, z5, tool0;
MoveL Offs(p0,368.5568,346.3328, 0), v100, z5, tool0;
MoveL Offs(p0,368.5109,346.21489999999994, 0), v100, z5, tool0;
MoveL Offs(p0,368.5016,346.0856, 0), v100, z5, tool0;
MoveL Offs(p0,368.5307,345.9467000000001, 0), v100, z5, tool0;
MoveL Offs(p0,368.6,345.8, 0), v100, z5, tool0;
MoveL Offs(p0,368.6,345.8, 0), v100, z5, tool0;
MoveJ Offs(p0,296.6,298.8, 10), v100, z1, tool0;
MoveL Offs(p0,296.38939999999997,295.4952, 0), v100, z5, tool0;
MoveL Offs(p0,296.34880000000004,294.5264, 0), v100, z5, tool0;
MoveL Offs(p0,296.325,293.65, 0), v100, z5, tool0;
MoveL Offs(p0,296.3192,292.8816, 0), v100, z5, tool0;
MoveL Offs(p0,296.3326,292.2368, 0), v100, z5, tool0;
MoveL Offs(p0,296.36640000000006,291.73120000000006, 0), v100, z5, tool0;
MoveL Offs(p0,297.43690000000004,291.9803, 0), v100, z5, tool0;
MoveL Offs(p0,297.76880000000006,292.8176, 0), v100, z5, tool0;
MoveL Offs(p0,298.0875,293.8625, 0), v100, z5, tool0;
MoveL Offs(p0,298.37919999999997,295.06640000000004, 0), v100, z5, tool0;
MoveL Offs(p0,298.63009999999997,296.3807, 0), v100, z5, tool0;
MoveL Offs(p0,298.82640000000004,297.7568, 0), v100, z5, tool0;
MoveL Offs(p0,298.95430000000005,299.14610000000005, 0), v100, z5, tool0;
MoveL Offs(p0,299.0,300.5, 0), v100, z5, tool0;
MoveL Offs(p0,298.61389999999994,304.76329999999996, 0), v100, z5, tool0;
MoveL Offs(p0,298.3568,305.2296, 0), v100, z5, tool0;
MoveL Offs(p0,298.0625,305.2375, 0), v100, z5, tool0;
MoveL Offs(p0,297.7472,304.7984, 0), v100, z5, tool0;
MoveL Offs(p0,297.4271,303.9237, 0), v100, z5, tool0;
MoveL Offs(p0,297.1184,302.62480000000005, 0), v100, z5, tool0;
MoveL Offs(p0,296.8373,300.91310000000004, 0), v100, z5, tool0;
MoveL Offs(p0,296.6,298.8, 0), v100, z5, tool0;
MoveL Offs(p0,296.6,298.8, 0), v100, z5, tool0;
MoveJ Offs(p0,295.4,271.1, 10), v100, z1, tool0;
MoveL Offs(p0,294.83510000000007,270.72990000000004, 0), v100, z5, tool0;
MoveL Offs(p0,294.2288000000001,270.2872000000001, 0), v100, z5, tool0;
MoveL Offs(p0,293.59369999999996,269.7833, 0), v100, z5, tool0;
MoveL Offs(p0,292.9424,269.2296, 0), v100, z5, tool0;
MoveL Offs(p0,292.2875,268.6375, 0), v100, z5, tool0;
MoveL Offs(p0,291.6416,268.01840000000004, 0), v100, z5, tool0;
MoveL Offs(p0,291.0173,267.3837, 0), v100, z5, tool0;
MoveL Offs(p0,290.42719999999997,266.74480000000005, 0), v100, z5, tool0;
MoveL Offs(p0,289.8839,266.11310000000003, 0), v100, z5, tool0;
MoveL Offs(p0,289.4,265.5, 0), v100, z5, tool0;
MoveL Offs(p0,288.12620000000004,264.12550000000005, 0), v100, z5, tool0;
MoveL Offs(p0,286.34960000000007,262.50800000000004, 0), v100, z5, tool0;
MoveL Offs(p0,284.1674,260.7165, 0), v100, z5, tool0;
MoveL Offs(p0,281.67680000000007,258.82000000000005, 0), v100, z5, tool0;
MoveL Offs(p0,278.975,256.8875, 0), v100, z5, tool0;
MoveL Offs(p0,276.1592,254.988, 0), v100, z5, tool0;
MoveL Offs(p0,273.3266,253.1905, 0), v100, z5, tool0;
MoveL Offs(p0,270.5744000000001,251.56400000000002, 0), v100, z5, tool0;
MoveL Offs(p0,267.9998,250.1775, 0), v100, z5, tool0;
MoveL Offs(p0,265.7,249.1, 0), v100, z5, tool0;
MoveL Offs(p0,264.83720000000005,248.7563000000001, 0), v100, z5, tool0;
MoveL Offs(p0,263.82560000000007,248.39040000000006, 0), v100, z5, tool0;
MoveL Offs(p0,262.6904,248.01009999999997, 0), v100, z5, tool0;
MoveL Offs(p0,261.4568,247.62320000000005, 0), v100, z5, tool0;
MoveL Offs(p0,260.15,247.2375, 0), v100, z5, tool0;
MoveL Offs(p0,258.7952,246.8608, 0), v100, z5, tool0;
MoveL Offs(p0,257.4176,246.5009, 0), v100, z5, tool0;
MoveL Offs(p0,256.0424,246.16559999999998, 0), v100, z5, tool0;
MoveL Offs(p0,254.69480000000004,245.86270000000005, 0), v100, z5, tool0;
MoveL Offs(p0,253.4,245.6, 0), v100, z5, tool0;
MoveL Offs(p0,251.33190000000005,245.17760000000004, 0), v100, z5, tool0;
MoveL Offs(p0,249.5512000000001,244.7408000000001, 0), v100, z5, tool0;
MoveL Offs(p0,248.03329999999997,244.27519999999998, 0), v100, z5, tool0;
MoveL Offs(p0,246.7536,243.76640000000003, 0), v100, z5, tool0;
MoveL Offs(p0,245.6875,243.2, 0), v100, z5, tool0;
MoveL Offs(p0,244.8104,242.5616, 0), v100, z5, tool0;
MoveL Offs(p0,244.09769999999997,241.83679999999998, 0), v100, z5, tool0;
MoveL Offs(p0,243.5248,241.0112, 0), v100, z5, tool0;
MoveL Offs(p0,243.06710000000004,240.0704, 0), v100, z5, tool0;
MoveL Offs(p0,242.7,239.0, 0), v100, z5, tool0;
MoveL Offs(p0,243.3608,235.08800000000002, 0), v100, z5, tool0;
MoveL Offs(p0,244.15,233.6375, 0), v100, z5, tool0;
MoveL Offs(p0,245.2632,231.872, 0), v100, z5, tool0;
MoveL Offs(p0,246.73760000000001,229.7285, 0), v100, z5, tool0;
MoveL Offs(p0,248.61040000000003,227.14400000000006, 0), v100, z5, tool0;
MoveL Offs(p0,250.9188,224.0555, 0), v100, z5, tool0;
MoveL Offs(p0,253.7,220.4, 0), v100, z5, tool0;
MoveL Offs(p0,255.3744,218.19650000000007, 0), v100, z5, tool0;
MoveL Offs(p0,257.13520000000005,215.87600000000006, 0), v100, z5, tool0;
MoveL Offs(p0,258.9488,213.4835, 0), v100, z5, tool0;
MoveL Offs(p0,260.7816,211.064, 0), v100, z5, tool0;
MoveL Offs(p0,262.6,208.6625, 0), v100, z5, tool0;
MoveL Offs(p0,264.3704,206.32399999999998, 0), v100, z5, tool0;
MoveL Offs(p0,266.05920000000003,204.0935, 0), v100, z5, tool0;
MoveL Offs(p0,267.63280000000003,202.01600000000002, 0), v100, z5, tool0;
MoveL Offs(p0,269.0576,200.1365, 0), v100, z5, tool0;
MoveL Offs(p0,270.3,198.5, 0), v100, z5, tool0;
MoveL Offs(p0,271.8041,196.41940000000005, 0), v100, z5, tool0;
MoveL Offs(p0,273.3328000000001,194.16720000000007, 0), v100, z5, tool0;
MoveL Offs(p0,274.9107,191.69779999999997, 0), v100, z5, tool0;
MoveL Offs(p0,276.5624,188.96560000000002, 0), v100, z5, tool0;
MoveL Offs(p0,278.3125,185.925, 0), v100, z5, tool0;
MoveL Offs(p0,280.18559999999997,182.53040000000001, 0), v100, z5, tool0;
MoveL Offs(p0,282.2063,178.7362, 0), v100, z5, tool0;
MoveL Offs(p0,284.3992,174.49680000000004, 0), v100, z5, tool0;
MoveL Offs(p0,286.7889,169.7666, 0), v100, z5, tool0;
MoveL Offs(p0,289.4,164.5, 0), v100, z5, tool0;
MoveL Offs(p0,291.4346,160.43290000000002, 0), v100, z5, tool0;
MoveL Offs(p0,293.43680000000006,156.49120000000005, 0), v100, z5, tool0;
MoveL Offs(p0,295.3742,152.73430000000002, 0), v100, z5, tool0;
MoveL Offs(p0,297.21440000000007,149.22160000000002, 0), v100, z5, tool0;
MoveL Offs(p0,298.925,146.0125, 0), v100, z5, tool0;
MoveL Offs(p0,300.47360000000003,143.16639999999998, 0), v100, z5, tool0;
MoveL Offs(p0,301.8278,140.7427, 0), v100, z5, tool0;
MoveL Offs(p0,302.95520000000005,138.80080000000004, 0), v100, z5, tool0;
MoveL Offs(p0,303.82340000000005,137.4001, 0), v100, z5, tool0;
MoveL Offs(p0,304.4,136.6, 0), v100, z5, tool0;
MoveL Offs(p0,305.07910000000004,135.9146, 0), v100, z5, tool0;
MoveL Offs(p0,305.69280000000015,135.35280000000003, 0), v100, z5, tool0;
MoveL Offs(p0,306.2657,134.90619999999998, 0), v100, z5, tool0;
MoveL Offs(p0,306.8224000000001,134.5664, 0), v100, z5, tool0;
MoveL Offs(p0,307.3875,134.325, 0), v100, z5, tool0;
MoveL Offs(p0,307.98560000000003,134.1736, 0), v100, z5, tool0;
MoveL Offs(p0,308.6413,134.1038, 0), v100, z5, tool0;
MoveL Offs(p0,309.3792,134.1072, 0), v100, z5, tool0;
MoveL Offs(p0,310.2239,134.17540000000002, 0), v100, z5, tool0;
MoveL Offs(p0,311.2,134.3, 0), v100, z5, tool0;
MoveL Offs(p0,314.0239,135.02980000000002, 0), v100, z5, tool0;
MoveL Offs(p0,318.0952000000001,136.57440000000003, 0), v100, z5, tool0;
MoveL Offs(p0,323.11330000000004,138.77659999999997, 0), v100, z5, tool0;
MoveL Offs(p0,328.7776,141.47920000000002, 0), v100, z5, tool0;
MoveL Offs(p0,334.7875,144.525, 0), v100, z5, tool0;
MoveL Offs(p0,340.8424,147.75680000000003, 0), v100, z5, tool0;
MoveL Offs(p0,346.64169999999996,151.0174, 0), v100, z5, tool0;
MoveL Offs(p0,351.8848,154.14960000000002, 0), v100, z5, tool0;
MoveL Offs(p0,356.2711,156.9962, 0), v100, z5, tool0;
MoveL Offs(p0,359.5,159.4, 0), v100, z5, tool0;
MoveL Offs(p0,361.132,160.8803, 0), v100, z5, tool0;
MoveL Offs(p0,362.3560000000001,162.33840000000006, 0), v100, z5, tool0;
MoveL Offs(p0,363.154,163.89010000000002, 0), v100, z5, tool0;
MoveL Offs(p0,363.508,165.65120000000002, 0), v100, z5, tool0;
MoveL Offs(p0,363.4,167.7375, 0), v100, z5, tool0;
MoveL Offs(p0,362.812,170.26479999999998, 0), v100, z5, tool0;
MoveL Offs(p0,361.726,173.34890000000001, 0), v100, z5, tool0;
MoveL Offs(p0,360.124,177.1056, 0), v100, z5, tool0;
MoveL Offs(p0,357.988,181.6507, 0), v100, z5, tool0;
MoveL Offs(p0,355.3,187.1, 0), v100, z5, tool0;
MoveL Offs(p0,352.83090000000004,192.0842, 0), v100, z5, tool0;
MoveL Offs(p0,350.48720000000014,196.72160000000005, 0), v100, z5, tool0;
MoveL Offs(p0,348.2143,201.1094, 0), v100, z5, tool0;
MoveL Offs(p0,345.9576,205.34480000000002, 0), v100, z5, tool0;
MoveL Offs(p0,343.6625,209.525, 0), v100, z5, tool0;
MoveL Offs(p0,341.2744,213.74719999999996, 0), v100, z5, tool0;
MoveL Offs(p0,338.7387,218.10859999999997, 0), v100, z5, tool0;
MoveL Offs(p0,336.0008,222.70640000000003, 0), v100, z5, tool0;
MoveL Offs(p0,333.0061,227.63780000000003, 0), v100, z5, tool0;
MoveL Offs(p0,329.7,233.0, 0), v100, z5, tool0;
MoveL Offs(p0,322.7024,244.3511, 0), v100, z5, tool0;
MoveL Offs(p0,317.0032000000001,253.4648000000001, 0), v100, z5, tool0;
MoveL Offs(p0,312.41279999999995,260.5517, 0), v100, z5, tool0;
MoveL Offs(p0,308.74160000000006,265.8224, 0), v100, z5, tool0;
MoveL Offs(p0,305.8,269.4875, 0), v100, z5, tool0;
MoveL Offs(p0,303.3984,271.7576, 0), v100, z5, tool0;
MoveL Offs(p0,301.3472,272.8433, 0), v100, z5, tool0;
MoveL Offs(p0,299.45680000000004,272.95520000000005, 0), v100, z5, tool0;
MoveL Offs(p0,297.5376,272.3039, 0), v100, z5, tool0;
MoveL Offs(p0,295.4,271.1, 0), v100, z5, tool0;
MoveL Offs(p0,295.4,271.1, 0), v100, z5, tool0;
MoveJ Offs(p0,303.0,269.0, 10), v100, z1, tool0;
MoveL Offs(p0,303.71950000000004,268.50350000000003, 0), v100, z5, tool0;
MoveL Offs(p0,304.3760000000001,267.80000000000007, 0), v100, z5, tool0;
MoveL Offs(p0,304.9665,266.89849999999996, 0), v100, z5, tool0;
MoveL Offs(p0,305.48800000000006,265.80800000000005, 0), v100, z5, tool0;
MoveL Offs(p0,305.9375,264.5375, 0), v100, z5, tool0;
MoveL Offs(p0,306.312,263.096, 0), v100, z5, tool0;
MoveL Offs(p0,306.6085,261.4925, 0), v100, z5, tool0;
MoveL Offs(p0,306.82400000000007,259.73600000000005, 0), v100, z5, tool0;
MoveL Offs(p0,306.95550000000003,257.8355, 0), v100, z5, tool0;
MoveL Offs(p0,307.0,255.8, 0), v100, z5, tool0;
MoveL Offs(p0,306.7592000000001,251.87120000000004, 0), v100, z5, tool0;
MoveL Offs(p0,306.4438,250.55479999999997, 0), v100, z5, tool0;
MoveL Offs(p0,305.98560000000003,249.66559999999998, 0), v100, z5, tool0;
MoveL Offs(p0,305.375,249.2, 0), v100, z5, tool0;
MoveL Offs(p0,304.6024,249.15439999999998, 0), v100, z5, tool0;
MoveL Offs(p0,303.6582,249.52519999999998, 0), v100, z5, tool0;
MoveL Offs(p0,302.53280000000007,250.30880000000002, 0), v100, z5, tool0;
MoveL Offs(p0,301.2166,251.5016, 0), v100, z5, tool0;
MoveL Offs(p0,299.7,253.1, 0), v100, z5, tool0;
MoveL Offs(p0,298.26540000000006,254.77850000000004, 0), v100, z5, tool0;
MoveL Offs(p0,297.0192000000001,256.34000000000003, 0), v100, z5, tool0;
MoveL Offs(p0,295.95779999999996,257.7935, 0), v100, z5, tool0;
MoveL Offs(p0,295.07759999999996,259.148, 0), v100, z5, tool0;
MoveL Offs(p0,294.375,260.4125, 0), v100, z5, tool0;
MoveL Offs(p0,293.8464,261.596, 0), v100, z5, tool0;
MoveL Offs(p0,293.4882,262.7075, 0), v100, z5, tool0;
MoveL Offs(p0,293.2968,263.75600000000003, 0), v100, z5, tool0;
MoveL Offs(p0,293.2686,264.7505, 0), v100, z5, tool0;
MoveL Offs(p0,293.4,265.7, 0), v100, z5, tool0;
MoveL Offs(p0,293.7876000000001,266.6969, 0), v100, z5, tool0;
MoveL Offs(p0,294.38880000000006,267.57920000000007, 0), v100, z5, tool0;
MoveL Offs(p0,295.1712,268.3343, 0), v100, z5, tool0;
MoveL Offs(p0,296.10240000000005,268.94960000000003, 0), v100, z5, tool0;
MoveL Offs(p0,297.15,269.4125, 0), v100, z5, tool0;
MoveL Offs(p0,298.28159999999997,269.71040000000005, 0), v100, z5, tool0;
MoveL Offs(p0,299.4648,269.8307, 0), v100, z5, tool0;
MoveL Offs(p0,300.66720000000004,269.7608, 0), v100, z5, tool0;
MoveL Offs(p0,301.8564,269.48810000000003, 0), v100, z5, tool0;
MoveL Offs(p0,303.0,269.0, 0), v100, z5, tool0;
MoveL Offs(p0,303.0,269.0, 0), v100, z5, tool0;
MoveJ Offs(p0,255.7,242.2, 10), v100, z1, tool0;
MoveL Offs(p0,256.29290000000003,241.62640000000005, 0), v100, z5, tool0;
MoveL Offs(p0,257.0232000000001,240.62320000000008, 0), v100, z5, tool0;
MoveL Offs(p0,257.8483,239.2768, 0), v100, z5, tool0;
MoveL Offs(p0,258.72560000000004,237.67360000000002, 0), v100, z5, tool0;
MoveL Offs(p0,259.6125,235.9, 0), v100, z5, tool0;
MoveL Offs(p0,260.46639999999996,234.0424, 0), v100, z5, tool0;
MoveL Offs(p0,261.2447,232.1872, 0), v100, z5, tool0;
MoveL Offs(p0,261.9048,230.4208, 0), v100, z5, tool0;
MoveL Offs(p0,262.4041,228.82960000000003, 0), v100, z5, tool0;
MoveL Offs(p0,262.7,227.5, 0), v100, z5, tool0;
MoveL Offs(p0,262.91360000000003,225.86880000000005, 0), v100, z5, tool0;
MoveL Offs(p0,262.9394,225.28869999999998, 0), v100, z5, tool0;
MoveL Offs(p0,262.25059999999996,224.1323, 0), v100, z5, tool0;
MoveL Offs(p0,261.82640000000004,224.04720000000003, 0), v100, z5, tool0;
MoveL Offs(p0,261.2798,224.00889999999998, 0), v100, z5, tool0;
MoveL Offs(p0,260.6,224.0, 0), v100, z5, tool0;
MoveL Offs(p0,258.70910000000003,224.44279999999998, 0), v100, z5, tool0;
MoveL Offs(p0,257.98720000000003,224.79360000000003, 0), v100, z5, tool0;
MoveL Offs(p0,257.2125,225.25, 0), v100, z5, tool0;
MoveL Offs(p0,256.3808,225.81439999999998, 0), v100, z5, tool0;
MoveL Offs(p0,255.4879,226.48919999999998, 0), v100, z5, tool0;
MoveL Offs(p0,254.52960000000002,227.2768, 0), v100, z5, tool0;
MoveL Offs(p0,253.50170000000003,228.17960000000002, 0), v100, z5, tool0;
MoveL Offs(p0,252.4,229.2, 0), v100, z5, tool0;
MoveL Offs(p0,251.1285000000001,230.43130000000002, 0), v100, z5, tool0;
MoveL Offs(p0,250.06400000000002,231.50240000000008, 0), v100, z5, tool0;
MoveL Offs(p0,249.1915,232.4391, 0), v100, z5, tool0;
MoveL Offs(p0,248.49600000000004,233.26720000000006, 0), v100, z5, tool0;
MoveL Offs(p0,247.9625,234.0125, 0), v100, z5, tool0;
MoveL Offs(p0,247.57599999999996,234.7008, 0), v100, z5, tool0;
MoveL Offs(p0,247.32150000000001,235.35789999999997, 0), v100, z5, tool0;
MoveL Offs(p0,247.18400000000003,236.00960000000003, 0), v100, z5, tool0;
MoveL Offs(p0,247.1485,236.6817, 0), v100, z5, tool0;
MoveL Offs(p0,247.2,237.4, 0), v100, z5, tool0;
MoveL Offs(p0,247.44880000000003,238.56040000000007, 0), v100, z5, tool0;
MoveL Offs(p0,247.93040000000005,239.62720000000013, 0), v100, z5, tool0;
MoveL Offs(p0,248.6076,240.5788, 0), v100, z5, tool0;
MoveL Offs(p0,249.4432,241.39359999999996, 0), v100, z5, tool0;
MoveL Offs(p0,250.4,242.05, 0), v100, z5, tool0;
MoveL Offs(p0,251.4408,242.52640000000002, 0), v100, z5, tool0;
MoveL Offs(p0,252.52839999999998,242.80120000000002, 0), v100, z5, tool0;
MoveL Offs(p0,253.62560000000002,242.85280000000003, 0), v100, z5, tool0;
MoveL Offs(p0,254.69520000000003,242.6596, 0), v100, z5, tool0;
MoveL Offs(p0,255.7,242.2, 0), v100, z5, tool0;
MoveL Offs(p0,255.7,242.2, 0), v100, z5, tool0;
MoveJ Offs(p0,327.9,224.3, 10), v100, z1, tool0;
MoveL Offs(p0,329.2559,222.9094, 0), v100, z5, tool0;
MoveL Offs(p0,331.1992000000001,220.37520000000004, 0), v100, z5, tool0;
MoveL Offs(p0,333.60329999999993,216.9038, 0), v100, z5, tool0;
MoveL Offs(p0,336.3416,212.70160000000004, 0), v100, z5, tool0;
MoveL Offs(p0,339.2875,207.975, 0), v100, z5, tool0;
MoveL Offs(p0,342.3144,202.9304, 0), v100, z5, tool0;
MoveL Offs(p0,345.2957,197.7742, 0), v100, z5, tool0;
MoveL Offs(p0,348.1048,192.71280000000002, 0), v100, z5, tool0;
MoveL Offs(p0,350.61510000000004,187.95260000000002, 0), v100, z5, tool0;
MoveL Offs(p0,352.7,183.7, 0), v100, z5, tool0;
MoveL Offs(p0,354.9,178.9, 0), v100, z5, tool0;
MoveL Offs(p0,352.7,180.5, 0), v100, z5, tool0;
MoveL Offs(p0,351.76490000000007,181.10910000000007, 0), v100, z5, tool0;
MoveL Offs(p0,350.8832000000001,181.55680000000007, 0), v100, z5, tool0;
MoveL Offs(p0,350.0603,181.8437, 0), v100, z5, tool0;
MoveL Offs(p0,349.3016,181.97039999999998, 0), v100, z5, tool0;
MoveL Offs(p0,348.6125,181.9375, 0), v100, z5, tool0;
MoveL Offs(p0,347.99839999999995,181.7456, 0), v100, z5, tool0;
MoveL Offs(p0,347.4647,181.3953, 0), v100, z5, tool0;
MoveL Offs(p0,347.01680000000005,180.88720000000004, 0), v100, z5, tool0;
MoveL Offs(p0,346.6601,180.2219, 0), v100, z5, tool0;
MoveL Offs(p0,346.4,179.4, 0), v100, z5, tool0;
MoveL Offs(p0,346.1855,178.02710000000005, 0), v100, z5, tool0;
MoveL Offs(p0,346.0760000000001,176.15680000000003, 0), v100, z5, tool0;
MoveL Offs(p0,346.0625,173.9217, 0), v100, z5, tool0;
MoveL Offs(p0,346.136,171.4544, 0), v100, z5, tool0;
MoveL Offs(p0,346.7885,163.9853, 0), v100, z5, tool0;
MoveL Offs(p0,347.12,161.9152, 0), v100, z5, tool0;
MoveL Offs(p0,347.4935,160.2759, 0), v100, z5, tool0;
MoveL Offs(p0,347.9,159.2, 0), v100, z5, tool0;
MoveL Offs(p0,348.15270000000004,158.6928, 0), v100, z5, tool0;
MoveL Offs(p0,348.3016000000001,158.23840000000004, 0), v100, z5, tool0;
MoveL Offs(p0,348.3329,157.8176, 0), v100, z5, tool0;
MoveL Offs(p0,348.2328000000001,157.4112, 0), v100, z5, tool0;
MoveL Offs(p0,347.5832,156.5648, 0), v100, z5, tool0;
MoveL Offs(p0,347.0061,156.0864, 0), v100, z5, tool0;
MoveL Offs(p0,346.2424,155.5456, 0), v100, z5, tool0;
MoveL Offs(p0,345.27830000000006,154.9232, 0), v100, z5, tool0;
MoveL Offs(p0,344.1,154.2, 0), v100, z5, tool0;
MoveL Offs(p0,343.1693,153.6271, 0), v100, z5, tool0;
MoveL Offs(p0,342.01840000000004,152.94080000000002, 0), v100, z5, tool0;
MoveL Offs(p0,340.67909999999995,152.1597, 0), v100, z5, tool0;
MoveL Offs(p0,339.18320000000006,151.3024, 0), v100, z5, tool0;
MoveL Offs(p0,337.5625,150.3875, 0), v100, z5, tool0;
MoveL Offs(p0,335.8488,149.43359999999998, 0), v100, z5, tool0;
MoveL Offs(p0,334.0739,148.45929999999998, 0), v100, z5, tool0;
MoveL Offs(p0,332.2696,147.4832, 0), v100, z5, tool0;
MoveL Offs(p0,330.46770000000004,146.5239, 0), v100, z5, tool0;
MoveL Offs(p0,328.7,145.6, 0), v100, z5, tool0;
MoveL Offs(p0,318.2,139.9, 0), v100, z5, tool0;
MoveL Offs(p0,317.6,143.5, 0), v100, z5, tool0;
MoveL Offs(p0,317.3938,144.31270000000004, 0), v100, z5, tool0;
MoveL Offs(p0,317.1264000000001,145.0816, 0), v100, z5, tool0;
MoveL Offs(p0,316.78459999999995,145.8229, 0), v100, z5, tool0;
MoveL Offs(p0,316.3552,146.55280000000002, 0), v100, z5, tool0;
MoveL Offs(p0,315.825,147.2875, 0), v100, z5, tool0;
MoveL Offs(p0,315.18080000000003,148.0432, 0), v100, z5, tool0;
MoveL Offs(p0,314.4094,148.8361, 0), v100, z5, tool0;
MoveL Offs(p0,313.49760000000003,149.68240000000003, 0), v100, z5, tool0;
MoveL Offs(p0,312.4322,150.59830000000002, 0), v100, z5, tool0;
MoveL Offs(p0,311.2,151.6, 0), v100, z5, tool0;
MoveL Offs(p0,309.39500000000004,152.98700000000002, 0), v100, z5, tool0;
MoveL Offs(p0,307.75200000000007,154.15200000000007, 0), v100, z5, tool0;
MoveL Offs(p0,306.25899999999996,155.10099999999997, 0), v100, z5, tool0;
MoveL Offs(p0,304.90400000000005,155.84000000000003, 0), v100, z5, tool0;
MoveL Offs(p0,303.675,156.375, 0), v100, z5, tool0;
MoveL Offs(p0,302.55999999999995,156.712, 0), v100, z5, tool0;
MoveL Offs(p0,301.54699999999997,156.857, 0), v100, z5, tool0;
MoveL Offs(p0,300.624,156.816, 0), v100, z5, tool0;
MoveL Offs(p0,299.77900000000005,156.595, 0), v100, z5, tool0;
MoveL Offs(p0,299.0,156.2, 0), v100, z5, tool0;
MoveL Offs(p0,298.13520000000005,155.97760000000005, 0), v100, z5, tool0;
MoveL Offs(p0,297.1936,156.6048, 0), v100, z5, tool0;
MoveL Offs(p0,296.625,157.3375, 0), v100, z5, tool0;
MoveL Offs(p0,295.95439999999996,158.4032, 0), v100, z5, tool0;
MoveL Offs(p0,295.1542,159.8421, 0), v100, z5, tool0;
MoveL Offs(p0,294.19680000000005,161.69440000000003, 0), v100, z5, tool0;
MoveL Offs(p0,293.05460000000005,164.0003, 0), v100, z5, tool0;
MoveL Offs(p0,291.7,166.8, 0), v100, z5, tool0;
MoveL Offs(p0,288.81800000000004,173.05730000000003, 0), v100, z5, tool0;
MoveL Offs(p0,286.4040000000001,178.66240000000002, 0), v100, z5, tool0;
MoveL Offs(p0,284.44599999999997,183.6651, 0), v100, z5, tool0;
MoveL Offs(p0,282.932,188.11520000000002, 0), v100, z5, tool0;
MoveL Offs(p0,281.85,192.0625, 0), v100, z5, tool0;
MoveL Offs(p0,281.188,195.5568, 0), v100, z5, tool0;
MoveL Offs(p0,280.934,198.6479, 0), v100, z5, tool0;
MoveL Offs(p0,281.076,201.3856, 0), v100, z5, tool0;
MoveL Offs(p0,281.602,203.8197, 0), v100, z5, tool0;
MoveL Offs(p0,282.5,206.0, 0), v100, z5, tool0;
MoveL Offs(p0,283.24370000000005,207.10250000000005, 0), v100, z5, tool0;
MoveL Offs(p0,284.3456000000001,208.28000000000003, 0), v100, z5, tool0;
MoveL Offs(p0,285.7319,209.4875, 0), v100, z5, tool0;
MoveL Offs(p0,287.32880000000006,210.68, 0), v100, z5, tool0;
MoveL Offs(p0,289.0625,211.8125, 0), v100, z5, tool0;
MoveL Offs(p0,290.8592,212.83999999999997, 0), v100, z5, tool0;
MoveL Offs(p0,292.6451,213.71749999999997, 0), v100, z5, tool0;
MoveL Offs(p0,294.3464,214.4, 0), v100, z5, tool0;
MoveL Offs(p0,295.8893,214.84250000000003, 0), v100, z5, tool0;
MoveL Offs(p0,297.2,215.0, 0), v100, z5, tool0;
MoveL Offs(p0,298.8288000000001,215.35680000000008, 0), v100, z5, tool0;
MoveL Offs(p0,299.7271999999999,215.7587, 0), v100, z5, tool0;
MoveL Offs(p0,300.6304,216.27040000000002, 0), v100, z5, tool0;
MoveL Offs(p0,301.5,216.8625, 0), v100, z5, tool0;
MoveL Offs(p0,302.2976,217.50560000000002, 0), v100, z5, tool0;
MoveL Offs(p0,302.9848,218.1703, 0), v100, z5, tool0;
MoveL Offs(p0,303.52320000000003,218.8272, 0), v100, z5, tool0;
MoveL Offs(p0,303.87440000000004,219.4469, 0), v100, z5, tool0;
MoveL Offs(p0,304.0,220.0, 0), v100, z5, tool0;
MoveL Offs(p0,304.2106,220.3355, 0), v100, z5, tool0;
MoveL Offs(p0,304.79680000000013,220.8360000000001, 0), v100, z5, tool0;
MoveL Offs(p0,305.6902,221.4625, 0), v100, z5, tool0;
MoveL Offs(p0,306.8224000000001,222.17600000000002, 0), v100, z5, tool0;
MoveL Offs(p0,308.125,222.9375, 0), v100, z5, tool0;
MoveL Offs(p0,309.52959999999996,223.708, 0), v100, z5, tool0;
MoveL Offs(p0,310.9678,224.44849999999997, 0), v100, z5, tool0;
MoveL Offs(p0,312.37120000000004,225.12000000000003, 0), v100, z5, tool0;
MoveL Offs(p0,313.6714,225.6835, 0), v100, z5, tool0;
MoveL Offs(p0,314.8,226.1, 0), v100, z5, tool0;
MoveL Offs(p0,316.03350000000006,226.39790000000002, 0), v100, z5, tool0;
MoveL Offs(p0,317.37200000000007,226.57520000000005, 0), v100, z5, tool0;
MoveL Offs(p0,318.78249999999997,226.6373, 0), v100, z5, tool0;
MoveL Offs(p0,320.232,226.58960000000002, 0), v100, z5, tool0;
MoveL Offs(p0,321.6875,226.4375, 0), v100, z5, tool0;
MoveL Offs(p0,324.4845,225.8417, 0), v100, z5, tool0;
MoveL Offs(p0,325.76000000000005,225.40879999999999, 0), v100, z5, tool0;
MoveL Offs(p0,326.9095,224.8931, 0), v100, z5, tool0;
MoveL Offs(p0,327.9,224.3, 0), v100, z5, tool0;
MoveL Offs(p0,327.9,224.3, 0), v100, z5, tool0;
MoveJ Offs(p0,353.4,176.9, 10), v100, z1, tool0;
MoveL Offs(p0,354.4150000000001,176.00390000000002, 0), v100, z5, tool0;
MoveL Offs(p0,355.35200000000003,175.01120000000003, 0), v100, z5, tool0;
MoveL Offs(p0,356.199,173.9453, 0), v100, z5, tool0;
MoveL Offs(p0,356.944,172.8296, 0), v100, z5, tool0;
MoveL Offs(p0,357.575,171.6875, 0), v100, z5, tool0;
MoveL Offs(p0,358.08,170.5424, 0), v100, z5, tool0;
MoveL Offs(p0,358.447,169.41770000000002, 0), v100, z5, tool0;
MoveL Offs(p0,358.66400000000004,168.33679999999998, 0), v100, z5, tool0;
MoveL Offs(p0,358.71900000000005,167.3231, 0), v100, z5, tool0;
MoveL Offs(p0,358.6,166.4, 0), v100, z5, tool0;
MoveL Offs(p0,358.23520000000013,165.58160000000004, 0), v100, z5, tool0;
MoveL Offs(p0,357.96729999999997,165.15439999999998, 0), v100, z5, tool0;
MoveL Offs(p0,357.6496,164.72480000000002, 0), v100, z5, tool0;
MoveL Offs(p0,357.2875,164.3, 0), v100, z5, tool0;
MoveL Offs(p0,356.8864,163.8872, 0), v100, z5, tool0;
MoveL Offs(p0,356.45169999999996,163.49360000000001, 0), v100, z5, tool0;
MoveL Offs(p0,355.9888,163.12640000000002, 0), v100, z5, tool0;
MoveL Offs(p0,355.5031,162.7928, 0), v100, z5, tool0;
MoveL Offs(p0,355.0,162.5, 0), v100, z5, tool0;
MoveL Offs(p0,354.2828,162.14900000000006, 0), v100, z5, tool0;
MoveL Offs(p0,353.6784000000001,161.87600000000003, 0), v100, z5, tool0;
MoveL Offs(p0,353.1676,161.68099999999998, 0), v100, z5, tool0;
MoveL Offs(p0,352.73120000000006,161.56400000000002, 0), v100, z5, tool0;
MoveL Offs(p0,352.35,161.525, 0), v100, z5, tool0;
MoveL Offs(p0,352.0048,161.56400000000002, 0), v100, z5, tool0;
MoveL Offs(p0,351.6764,161.68099999999998, 0), v100, z5, tool0;
MoveL Offs(p0,351.3456,161.87600000000003, 0), v100, z5, tool0;
MoveL Offs(p0,350.9932,162.14900000000003, 0), v100, z5, tool0;
MoveL Offs(p0,350.07950000000005,163.2262, 0), v100, z5, tool0;
MoveL Offs(p0,349.6040000000001,164.22960000000003, 0), v100, z5, tool0;
MoveL Offs(p0,349.1825,165.45739999999998, 0), v100, z5, tool0;
MoveL Offs(p0,348.824,166.85680000000002, 0), v100, z5, tool0;
MoveL Offs(p0,348.5375,168.375, 0), v100, z5, tool0;
MoveL Offs(p0,348.332,169.95919999999998, 0), v100, z5, tool0;
MoveL Offs(p0,348.2165,171.55659999999997, 0), v100, z5, tool0;
MoveL Offs(p0,348.2,173.11440000000002, 0), v100, z5, tool0;
MoveL Offs(p0,348.29150000000004,174.5798, 0), v100, z5, tool0;
MoveL Offs(p0,348.5,175.9, 0), v100, z5, tool0;
MoveL Offs(p0,348.73710000000005,176.90270000000004, 0), v100, z5, tool0;
MoveL Offs(p0,348.98080000000004,177.69360000000006, 0), v100, z5, tool0;
MoveL Offs(p0,349.2497,178.2769, 0), v100, z5, tool0;
MoveL Offs(p0,349.56239999999997,178.65680000000003, 0), v100, z5, tool0;
MoveL Offs(p0,349.9375,178.8375, 0), v100, z5, tool0;
MoveL Offs(p0,350.3936,178.82319999999999, 0), v100, z5, tool0;
MoveL Offs(p0,350.9493,178.6181, 0), v100, z5, tool0;
MoveL Offs(p0,351.6232,178.2264, 0), v100, z5, tool0;
MoveL Offs(p0,352.43390000000005,177.65230000000003, 0), v100, z5, tool0;
MoveL Offs(p0,353.4,176.9, 0), v100, z5, tool0;
MoveL Offs(p0,353.4,176.9, 0), v100, z5, tool0;
MoveJ Offs(p0,308.9,150.0, 10), v100, z1, tool0;
MoveL Offs(p0,310.41,148.75590000000003, 0), v100, z5, tool0;
MoveL Offs(p0,311.64400000000006,147.59520000000003, 0), v100, z5, tool0;
MoveL Offs(p0,312.608,146.50529999999998, 0), v100, z5, tool0;
MoveL Offs(p0,313.308,145.4736, 0), v100, z5, tool0;
MoveL Offs(p0,313.75,144.4875, 0), v100, z5, tool0;
MoveL Offs(p0,313.93999999999994,143.53439999999998, 0), v100, z5, tool0;
MoveL Offs(p0,313.884,142.6017, 0), v100, z5, tool0;
MoveL Offs(p0,313.588,141.67680000000001, 0), v100, z5, tool0;
MoveL Offs(p0,313.05800000000005,140.7471, 0), v100, z5, tool0;
MoveL Offs(p0,312.3,139.8, 0), v100, z5, tool0;
MoveL Offs(p0,312.0132000000001,139.50660000000002, 0), v100, z5, tool0;
MoveL Offs(p0,311.6976,139.22880000000004, 0), v100, z5, tool0;
MoveL Offs(p0,311.36039999999997,138.9702, 0), v100, z5, tool0;
MoveL Offs(p0,311.0088,138.7344, 0), v100, z5, tool0;
MoveL Offs(p0,310.65,138.525, 0), v100, z5, tool0;
MoveL Offs(p0,310.2912,138.3456, 0), v100, z5, tool0;
MoveL Offs(p0,309.93960000000004,138.1998, 0), v100, z5, tool0;
MoveL Offs(p0,309.60240000000005,138.09120000000001, 0), v100, z5, tool0;
MoveL Offs(p0,309.28679999999997,138.02339999999998, 0), v100, z5, tool0;
MoveL Offs(p0,309.0,138.0, 0), v100, z5, tool0;
MoveL Offs(p0,307.40480000000014,138.47600000000006, 0), v100, z5, tool0;
MoveL Offs(p0,306.56370000000004,139.0395, 0), v100, z5, tool0;
MoveL Offs(p0,305.7184,139.792, 0), v100, z5, tool0;
MoveL Offs(p0,304.8875,140.7125, 0), v100, z5, tool0;
MoveL Offs(p0,304.08959999999996,141.78, 0), v100, z5, tool0;
MoveL Offs(p0,303.3433,142.9735, 0), v100, z5, tool0;
MoveL Offs(p0,302.66720000000004,144.27200000000002, 0), v100, z5, tool0;
MoveL Offs(p0,302.0799,145.6545, 0), v100, z5, tool0;
MoveL Offs(p0,301.6,147.1, 0), v100, z5, tool0;
MoveL Offs(p0,301.016,149.31150000000002, 0), v100, z5, tool0;
MoveL Offs(p0,300.7080000000001,151.08800000000002, 0), v100, z5, tool0;
MoveL Offs(p0,300.6820000000001,152.43249999999998, 0), v100, z5, tool0;
MoveL Offs(p0,300.944,153.348, 0), v100, z5, tool0;
MoveL Offs(p0,302.35600000000005,153.904, 0), v100, z5, tool0;
MoveL Offs(p0,303.518,153.5505, 0), v100, z5, tool0;
MoveL Offs(p0,304.992,152.78000000000003, 0), v100, z5, tool0;
MoveL Offs(p0,306.784,151.59550000000002, 0), v100, z5, tool0;
MoveL Offs(p0,308.9,150.0, 0), v100, z5, tool0;
MoveL Offs(p0,308.9,150.0, 0), v100, z5, tool0;
MoveJ Offs(p0,271.6,278.4, 10), v100, z1, tool0;
MoveL Offs(p0,271.1267,277.86, 0), v100, z5, tool0;
MoveL Offs(p0,270.7296000000001,277.22400000000005, 0), v100, z5, tool0;
MoveL Offs(p0,270.4129,276.52799999999996, 0), v100, z5, tool0;
MoveL Offs(p0,270.1808,275.80800000000005, 0), v100, z5, tool0;
MoveL Offs(p0,270.0375,275.1, 0), v100, z5, tool0;
MoveL Offs(p0,269.9872,274.43999999999994, 0), v100, z5, tool0;
MoveL Offs(p0,270.0341,273.864, 0), v100, z5, tool0;
MoveL Offs(p0,270.18240000000003,273.408, 0), v100, z5, tool0;
MoveL Offs(p0,270.4363,273.108, 0), v100, z5, tool0;
MoveL Offs(p0,270.8,273.0, 0), v100, z5, tool0;
MoveL Offs(p0,271.98640000000006,273.5880000000001, 0), v100, z5, tool0;
MoveL Offs(p0,272.75660000000005,274.2285, 0), v100, z5, tool0;
MoveL Offs(p0,273.5712,275.01599999999996, 0), v100, z5, tool0;
MoveL Offs(p0,274.375,275.8875, 0), v100, z5, tool0;
MoveL Offs(p0,275.1128,276.78000000000003, 0), v100, z5, tool0;
MoveL Offs(p0,275.7294,277.6305, 0), v100, z5, tool0;
MoveL Offs(p0,276.16960000000006,278.37600000000003, 0), v100, z5, tool0;
MoveL Offs(p0,276.3782,278.95349999999996, 0), v100, z5, tool0;
MoveL Offs(p0,276.3,279.3, 0), v100, z5, tool0;
MoveL Offs(p0,275.94430000000006,279.61230000000006, 0), v100, z5, tool0;
MoveL Offs(p0,275.5424000000001,279.83040000000005, 0), v100, z5, tool0;
MoveL Offs(p0,275.10209999999995,279.9561, 0), v100, z5, tool0;
MoveL Offs(p0,274.63120000000004,279.99120000000005, 0), v100, z5, tool0;
MoveL Offs(p0,274.1375,279.9375, 0), v100, z5, tool0;
MoveL Offs(p0,273.6288,279.79679999999996, 0), v100, z5, tool0;
MoveL Offs(p0,273.11289999999997,279.5709, 0), v100, z5, tool0;
MoveL Offs(p0,272.0907,278.87070000000006, 0), v100, z5, tool0;
MoveL Offs(p0,271.6,278.4, 0), v100, z5, tool0;
MoveL Offs(p0,271.6,278.4, 0), v100, z5, tool0;
MoveJ Offs(p0,247.8,264.9, 10), v100, z1, tool0;
MoveL Offs(p0,247.27249999999998,264.56090000000006, 0), v100, z5, tool0;
MoveL Offs(p0,246.8320000000001,264.15520000000004, 0), v100, z5, tool0;
MoveL Offs(p0,246.4815,263.7003, 0), v100, z5, tool0;
MoveL Offs(p0,246.22400000000002,263.21360000000004, 0), v100, z5, tool0;
MoveL Offs(p0,246.0625,262.7125, 0), v100, z5, tool0;
MoveL Offs(p0,246.0,262.21439999999996, 0), v100, z5, tool0;
MoveL Offs(p0,246.0395,261.7367, 0), v100, z5, tool0;
MoveL Offs(p0,246.18400000000003,261.2968, 0), v100, z5, tool0;
MoveL Offs(p0,246.43650000000002,260.9121, 0), v100, z5, tool0;
MoveL Offs(p0,246.8,260.6, 0), v100, z5, tool0;
MoveL Offs(p0,248.325,260.9125, 0), v100, z5, tool0;
MoveL Offs(p0,248.7944,261.104, 0), v100, z5, tool0;
MoveL Offs(p0,249.29619999999994,261.33149999999995, 0), v100, z5, tool0;
MoveL Offs(p0,249.82080000000005,261.592, 0), v100, z5, tool0;
MoveL Offs(p0,250.35860000000002,261.88250000000005, 0), v100, z5, tool0;
MoveL Offs(p0,250.9,262.2, 0), v100, z5, tool0;
MoveL Offs(p0,251.56339999999994,262.65380000000005, 0), v100, z5, tool0;
MoveL Offs(p0,252.1152000000001,263.05840000000006, 0), v100, z5, tool0;
MoveL Offs(p0,252.5578,263.4186, 0), v100, z5, tool0;
MoveL Offs(p0,252.89360000000002,263.7392000000001, 0), v100, z5, tool0;
MoveL Offs(p0,253.125,264.025, 0), v100, z5, tool0;
MoveL Offs(p0,253.25439999999998,264.28080000000006, 0), v100, z5, tool0;
MoveL Offs(p0,253.2842,264.5114, 0), v100, z5, tool0;
MoveL Offs(p0,253.2168,264.7216, 0), v100, z5, tool0;
MoveL Offs(p0,253.05460000000002,264.9162, 0), v100, z5, tool0;
MoveL Offs(p0,252.8,265.1, 0), v100, z5, tool0;
MoveL Offs(p0,252.30360000000002,265.39680000000004, 0), v100, z5, tool0;
MoveL Offs(p0,251.82880000000006,265.62640000000005, 0), v100, z5, tool0;
MoveL Offs(p0,251.3672,265.7876, 0), v100, z5, tool0;
MoveL Offs(p0,250.91040000000004,265.87919999999997, 0), v100, z5, tool0;
MoveL Offs(p0,250.45,265.9, 0), v100, z5, tool0;
MoveL Offs(p0,249.9776,265.8488, 0), v100, z5, tool0;
MoveL Offs(p0,249.4848,265.72439999999995, 0), v100, z5, tool0;
MoveL Offs(p0,248.9632,265.52560000000005, 0), v100, z5, tool0;
MoveL Offs(p0,247.8,264.9, 0), v100, z5, tool0;
MoveL Offs(p0,247.8,264.9, 0), v100, z5, tool0;
MoveJ Offs(p0,214.0,259.2, 10), v100, z1, tool0;
MoveL Offs(p0,214.22640000000007,258.8144000000001, 0), v100, z5, tool0;
MoveL Offs(p0,214.49409999999997,258.5241, 0), v100, z5, tool0;
MoveL Offs(p0,214.8512,258.17920000000004, 0), v100, z5, tool0;
MoveL Offs(p0,215.2875,257.7875, 0), v100, z5, tool0;
MoveL Offs(p0,215.7928,257.3568, 0), v100, z5, tool0;
MoveL Offs(p0,216.3569,256.89489999999995, 0), v100, z5, tool0;
MoveL Offs(p0,216.96960000000004,256.40960000000007, 0), v100, z5, tool0;
MoveL Offs(p0,217.6207,255.9087, 0), v100, z5, tool0;
MoveL Offs(p0,218.3,255.4, 0), v100, z5, tool0;
MoveL Offs(p0,219.65200000000004,254.4353, 0), v100, z5, tool0;
MoveL Offs(p0,220.99200000000005,253.58640000000005, 0), v100, z5, tool0;
MoveL Offs(p0,222.296,252.8611, 0), v100, z5, tool0;
MoveL Offs(p0,223.54000000000002,252.2672, 0), v100, z5, tool0;
MoveL Offs(p0,224.7,251.8125, 0), v100, z5, tool0;
MoveL Offs(p0,225.752,251.5048, 0), v100, z5, tool0;
MoveL Offs(p0,226.67199999999997,251.35189999999997, 0), v100, z5, tool0;
MoveL Offs(p0,227.43600000000006,251.3616, 0), v100, z5, tool0;
MoveL Offs(p0,228.02000000000004,251.54170000000005, 0), v100, z5, tool0;
MoveL Offs(p0,228.4,251.9, 0), v100, z5, tool0;
MoveL Offs(p0,227.9875,252.7375, 0), v100, z5, tool0;
MoveL Offs(p0,227.6944,252.908, 0), v100, z5, tool0;
MoveL Offs(p0,227.34369999999998,253.0725, 0), v100, z5, tool0;
MoveL Offs(p0,226.94080000000002,253.228, 0), v100, z5, tool0;
MoveL Offs(p0,226.49110000000002,253.37150000000003, 0), v100, z5, tool0;
MoveL Offs(p0,226.0,253.5, 0), v100, z5, tool0;
MoveL Offs(p0,225.03040000000004,253.7728000000001, 0), v100, z5, tool0;
MoveL Offs(p0,224.63109999999998,253.93019999999996, 0), v100, z5, tool0;
MoveL Offs(p0,224.29120000000003,254.0984, 0), v100, z5, tool0;
MoveL Offs(p0,224.0125,254.275, 0), v100, z5, tool0;
MoveL Offs(p0,223.7968,254.4576, 0), v100, z5, tool0;
MoveL Offs(p0,223.64590000000004,254.6438, 0), v100, z5, tool0;
MoveL Offs(p0,223.5616,254.8312, 0), v100, z5, tool0;
MoveL Offs(p0,223.54569999999998,255.0174, 0), v100, z5, tool0;
MoveL Offs(p0,223.6,255.2, 0), v100, z5, tool0;
MoveL Offs(p0,223.825,255.6293, 0), v100, z5, tool0;
MoveL Offs(p0,223.84000000000006,255.72160000000002, 0), v100, z5, tool0;
MoveL Offs(p0,223.825,255.7875, 0), v100, z5, tool0;
MoveL Offs(p0,223.3,255.7, 0), v100, z5, tool0;
MoveL Offs(p0,221.45229999999998,256.0186, 0), v100, z5, tool0;
MoveL Offs(p0,220.58960000000002,256.4072, 0), v100, z5, tool0;
MoveL Offs(p0,219.7125,256.875, 0), v100, z5, tool0;
MoveL Offs(p0,218.8864,257.3848, 0), v100, z5, tool0;
MoveL Offs(p0,218.17669999999998,257.8994, 0), v100, z5, tool0;
MoveL Offs(p0,217.64880000000002,258.38160000000005, 0), v100, z5, tool0;
MoveL Offs(p0,217.3681,258.7942, 0), v100, z5, tool0;
MoveL Offs(p0,217.4,259.1, 0), v100, z5, tool0;
MoveL Offs(p0,217.1875,259.475, 0), v100, z5, tool0;
MoveL Offs(p0,217.0112,259.532, 0), v100, z5, tool0;
MoveL Offs(p0,216.80010000000001,259.58299999999997, 0), v100, z5, tool0;
MoveL Offs(p0,216.55839999999998,259.62800000000004, 0), v100, z5, tool0;
MoveL Offs(p0,216.29030000000003,259.66700000000003, 0), v100, z5, tool0;
MoveL Offs(p0,216.0,259.7, 0), v100, z5, tool0;
MoveL Offs(p0,214.10240000000005,259.4152, 0), v100, z5, tool0;
MoveL Offs(p0,214.0263,259.3139, 0), v100, z5, tool0;
MoveL Offs(p0,214.0,259.2, 0), v100, z5, tool0;
MoveL Offs(p0,214.0,259.2, 0), v100, z5, tool0;
MoveJ Offs(p0,462.5,184.1, 10), v100, z1, tool0;
MoveL Offs(p0,462.8,182.6, 0), v100, z5, tool0;
MoveL Offs(p0,463.6001,182.8961, 0), v100, z5, tool0;
MoveL Offs(p0,463.6544,183.0704, 0), v100, z5, tool0;
MoveL Offs(p0,463.68829999999997,183.2723, 0), v100, z5, tool0;
MoveL Offs(p0,463.7,183.5, 0), v100, z5, tool0;
MoveL Offs(p0,463.4375,184.925, 0), v100, z5, tool0;
MoveL Offs(p0,463.31119999999993,184.94, 0), v100, z5, tool0;
MoveL Offs(p0,463.1561,184.865, 0), v100, z5, tool0;
MoveL Offs(p0,462.9704,184.7, 0), v100, z5, tool0;
MoveL Offs(p0,462.7523,184.445, 0), v100, z5, tool0;
MoveL Offs(p0,462.5,184.1, 0), v100, z5, tool0;
MoveL Offs(p0,462.5,184.1, 0), v100, z5, tool0;
    ENDPROC
ENDMODULE
